Staubli VAL3: main.pgx

public program main()
  local bool l_bSave
  local num l_nIndex
  local string l_sEvent
  local bool l_bFound
  local InstrItem l_iInstr
  local string l_sPath
  local bool l_bUnreached
  local string l_sMessage
begin
  // INIT
  call onStart()
  // LOOP UNTIL nKey=255
  do
    // refresh
    call refresh()
    nKey=getKey()
    call use:listevent(nKey,nId,sEvent)
    nSelected=nId
    nView=use:nView
    // get the index
    if find(left(sEvent,1)," ")!=-1
      l_sEvent=right(sEvent,len(sEvent)-1)
    else
      l_sEvent=sEvent
    endIf
    toNum(l_sEvent,l_nIndex,l_bFound)
    if l_bFound
      nIndex=l_nIndex-1
    endIf
    // check for the moveHold
    call prog:getItem(l_iInstr,nIndex)
    call saveData:getPathInstr(l_iInstr.sType,l_sPath)
    if find(l_sPath,"trajectory")!=-1
      call goTo(l_bUnreached,l_iInstr)
      if l_bUnreached
        // show the message out of range
        call language:message(l_sMessage,-5)
        call use:timerDialog(l_sMessage,1)
        l_bUnreached=false
      endIf
    endIf
    // key capture
    switch nKey
      case 259
        // TAB-> ENLARGE
        bLarge=!bLarge
        call use:setView(bLarge)
      break
      case 263
        // backSpace
        if l_bFound
          call onBackEvent(l_bSave)
        endIf
      break
      case 271
        // Simulation
        if l_bFound
          call onF1Event()
        endIf
      break
      case 272
        call onF2Event(l_bSave)
      break
      case 273
        // INPUT OUTPUT
        call onF3Event(l_bSave)
      break
      case 274
        // PASTE
        call onF4Event(l_bSave)
      break
      case 275
        // SELECT_UNSELECT
        if l_bFound
          call onF5Event()
        endIf
      break
      case 276
        // DELETE
        if l_bFound
          call onF6Event(l_bSave)
        endIf
      break
      case 277
        //INSERT
        if l_bFound or l_sEvent==""
          call onF7Event(l_bSave)
        endIf
      break
      case 278
        // SAVE
        call onF8Event(l_bSave)
      break
      case 270
        if l_bFound
          // EDIT THE FIELD
          call onEnterEvent(l_bSave)
        endIf
      break
      case 255
        // exit??
        // on Exit
        call onExit(l_bSave)
      break
    endSwitch
    //release the resource
    delay(0.1)
  until bExit
  //
  // reset
  //
  bExit=false
end
